Fanuc KAREL source: MP0076.KL

-- PROVISIONAL review KL for V1013-1; original PC SHA256 63394ae713bb27732670cc4f87244f88d477293601d4723bb145fc52e67aba3b
-- Incomplete behavior may be omitted. Consult companion uncertainty JSON. Do not deploy.
PROGRAM MP0076
%NOLOCKGROUP
-- UNRESOLVED_LOCAL_POOL 8 cells at code offset 65; source declarations unknown
-- DIRECT_LOCAL_WORD_ACCESS alone does not prove INTEGER, REAL, or BOOLEAN
BEGIN
  -- UNRESOLVED_PC offsets 0-1; opcodes 7B
  -- UNRESOLVED_PC offsets 6-18; opcodes 2D,9D,52,7F
  -- UNRESOLVED_PC offsets 23-28; opcodes 7F,7B
  -- UNRESOLVED_PC offsets 33-49; opcodes 2D,2E,69,7F
  -- UNRESOLVED_PC offsets 54-70; opcodes 7F,2B,2C,7B
  -- UNRESOLVED_PC offsets 75-86; opcodes 2E,23
  -- UNRESOLVED_PC offsets 91-102; opcodes 2E,23
  -- UNRESOLVED_PC offsets 107-118; opcodes 2E,23
  -- UNRESOLVED_PC offsets 123-134; opcodes 2E,23
  -- UNRESOLVED_PC offsets 139-150; opcodes 2E,23
  -- UNRESOLVED_PC offsets 155-166; opcodes 2E,23
  -- UNRESOLVED_PC offsets 171-185; opcodes 2E,22,9D,33,35
  -- UNRESOLVED_PC offsets 190-216; opcodes 22,9D,33,34,21,64,29,64,29,6C,23
  -- UNRESOLVED_PC offsets 221-225; opcodes 7F
  -- UNRESOLVED_PC offsets 230-246; opcodes 27,27,2E,27,2E,AA
  -- UNRESOLVED_PC offsets 251-255; opcodes 7F
END MP0076
